PROGRAM PANEL
VAR
	START:BOOL;
	STOP:BOOL;
	HOME:BOOL;
	WRITE:BOOL;
	M00:BOOL;
	M01:BOOL;
	TON_0: TON;
	
	
END_VAR
VAR // added by the converter: edge detectors and wires of the graphical bodies
    _w1, _w2, _w3, _w4, _w5 : BOOL;
END_VAR

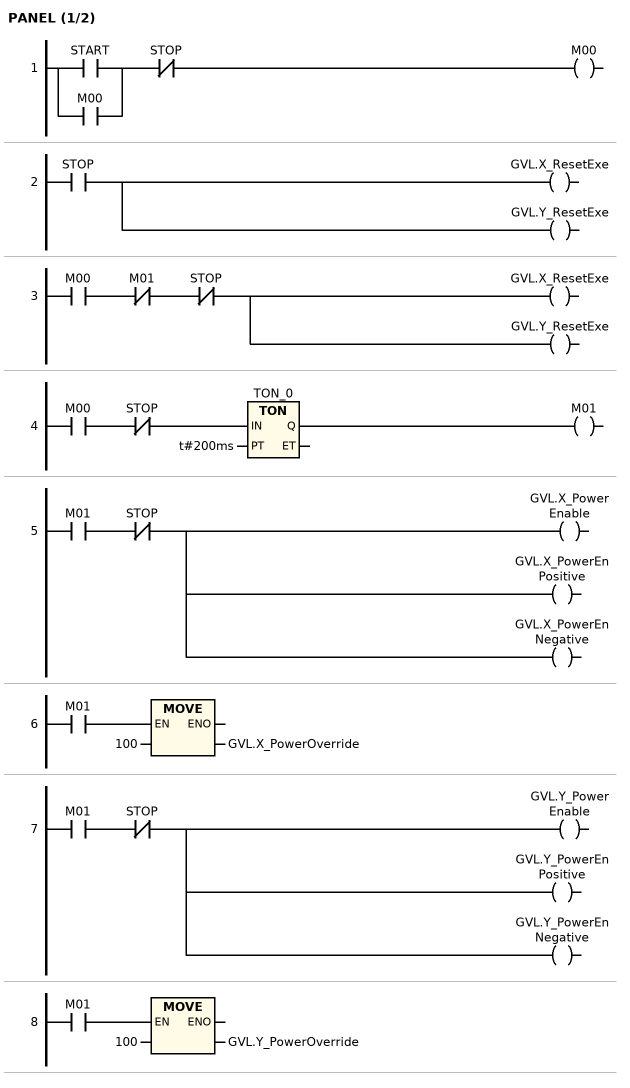
// NETWORK 1
M00 := (START OR M00) AND NOT STOP;

// NETWORK 2
GVL.X_ResetExe := STOP;
GVL.Y_ResetExe := STOP;

// NETWORK 3
_w1 := M00 AND NOT M01 AND NOT STOP;
GVL.X_ResetExe := _w1;
GVL.Y_ResetExe := _w1;

// NETWORK 4
TON_0(IN := M00 AND NOT STOP, PT := t#200ms); // TON
M01 := TON_0.Q;

// NETWORK 5
_w2 := M01 AND NOT STOP;
GVL.X_PowerEnable := _w2;
GVL.X_PowerEnPositive := _w2;
GVL.X_PowerEnNegative := _w2;

// NETWORK 6
IF M01 THEN GVL.X_PowerOverride := 100; END_IF

// NETWORK 7
_w3 := M01 AND NOT STOP;
GVL.Y_PowerEnable := _w3;
GVL.Y_PowerEnPositive := _w3;
GVL.Y_PowerEnNegative := _w3;

// NETWORK 8
IF M01 THEN GVL.Y_PowerOverride := 100; END_IF

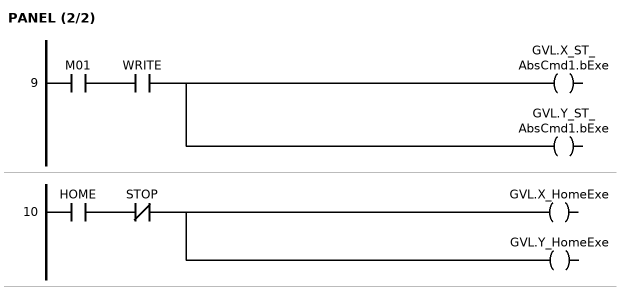
// NETWORK 9
_w4 := M01 AND WRITE;
GVL.X_ST_AbsCmd1.bExe := _w4;
GVL.Y_ST_AbsCmd1.bExe := _w4;

// NETWORK 10
_w5 := HOME AND NOT STOP;
GVL.X_HomeExe := _w5;
GVL.Y_HomeExe := _w5;

END_PROGRAM

(* stored: Version 1.1.0.1, ProductVersion 3.1.4024.13
   POU PANEL: Id {8a2f159b-bec7-4b77-8eee-0052e44aeef5}, SpecialFunc None *)
